PROGRAM MAIN
VAR
	iCounterValueDoubleCheckEL5101		AT%I*			:UDINT;
	bResetCounterEL5101					AT%Q*			:BOOL;
	iSetCounterValueEL5101ForReset		AT%Q*			:UDINT;
	
	bResetEL5101										:bool;
END_VAR

bResetCounterEL5101:=FALSE;

IF bResetEL5101 THEN
	bResetCounterEL5101:=TRUE;
	iSetCounterValueEL5101ForReset:=0;
	bResetEL5101:=FALSE;
END_IF

END_PROGRAM

(* stored: Version 1.1.0.1, ProductVersion 3.1.4024.11
   POU MAIN: Id {c46370cb-00d4-4024-9723-0e4e960bd11c}, SpecialFunc None *)
